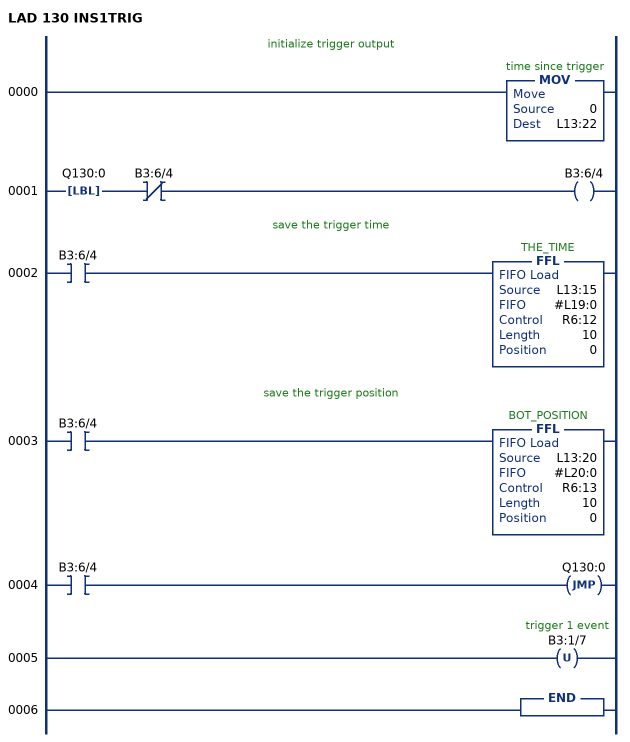
% Rung: 0 %
% initialize trigger output %
SOR MOV 0 L13:22 EOR
%   L13:22  "time since trigger" %
% Rung: 1 %
SOR LBL Q130:0 XIO B3:6/4 OTE B3:6/4 EOR
% Rung: 2 %
% save the trigger time %
SOR XIC B3:6/4 FFL L13:15 #L19:0 R6:12 10 0 EOR
%   L13:15  THE_TIME %
% Rung: 3 %
% save the trigger position %
SOR XIC B3:6/4 FFL L13:20 #L20:0 R6:13 10 0 EOR
%   L13:20  BOT_POSITION %
% Rung: 4 %
SOR XIC B3:6/4 JMP Q130:0 EOR
% Rung: 5 %
SOR OTU B3:1/7 EOR
%   B3:1/7  "trigger 1 event" %
% Rung: 6 %
SOR END EOR

LADDER 131 "XFER"
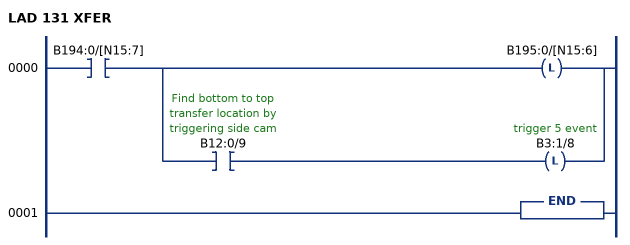
% Rung: 0 %
SOR XIC B194:0/[N15:7] BST OTL B195:0/[N15:6] NXB XIC B12:0/9 OTL B3:1/8 BND EOR
%   N15:7  XFER_OUT_LOC %
%   N15:6  XFER_IN_LOC %
%   B12:0/9  "Find bottom to top transfer location by triggering side cam" %
%   B3:1/8  "trigger 5 event" %
% Rung: 1 %
SOR END EOR

LADDER 140 "TOPOPTIC"
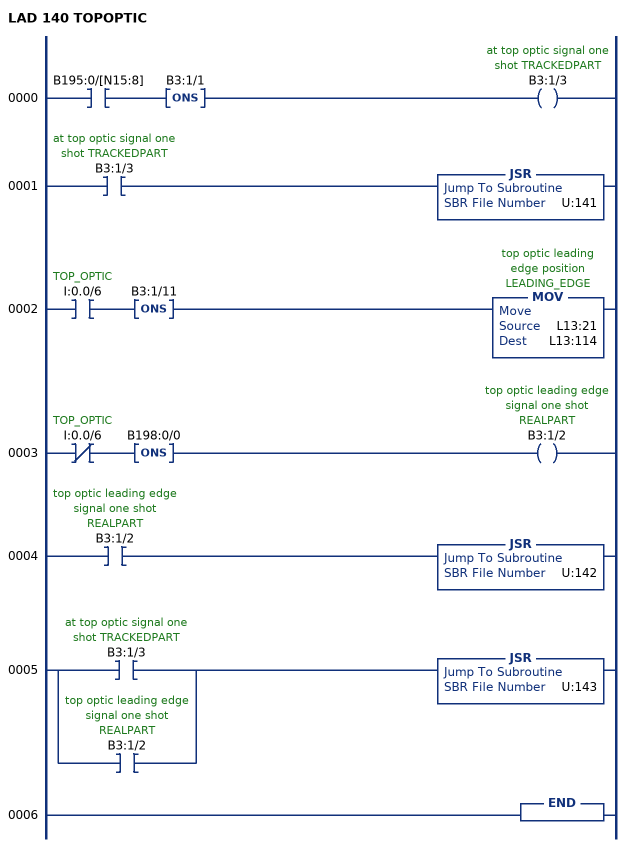
% Rung: 0 %
SOR XIC B195:0/[N15:8] ONS B3:1/1 OTE B3:1/3 EOR
%   N15:8  TOP_OPTIC_LOC %
%   B3:1/3  TRACKEDPART  "at top optic signal one shot" %
% Rung: 1 %
SOR XIC B3:1/3 JSR U:141 EOR
%   B3:1/3  TRACKEDPART  "at top optic signal one shot" %
% Rung: 2 %
SOR XIC I:0.0/6 ONS B3:1/11 MOV L13:21 L13:114 EOR
%   I:0.0/6  TOP_OPTIC %
%   L13:21  TOP_POSITION %
%   L13:114  LEADING_EDGE  "top optic leading edge position" %
% Rung: 3 %
SOR XIO I:0.0/6 ONS B198:0/0 OTE B3:1/2 EOR
%   I:0.0/6  TOP_OPTIC %
%   B3:1/2  REALPART  "top optic leading edge signal one shot" %
% Rung: 4 %
SOR XIC B3:1/2 JSR U:142 EOR
%   B3:1/2  REALPART  "top optic leading edge signal one shot" %
% Rung: 5 %
SOR BST XIC B3:1/3 NXB XIC B3:1/2 BND JSR U:143 EOR
%   B3:1/3  TRACKEDPART  "at top optic signal one shot" %
%   B3:1/2  REALPART  "top optic leading edge signal one shot" %
% Rung: 6 %
SOR END EOR

LADDER 141 "TOPOPVERT"
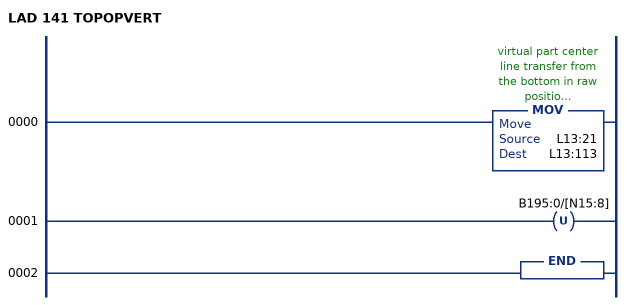
% Rung: 0 %
SOR MOV L13:21 L13:113 EOR
%   L13:21  TOP_POSITION %
%   L13:113  VERTUAL_PT_RAW_CL  "virtual part center line transfer from the bottom in raw position" %
% Rung: 1 %
SOR OTU B195:0/[N15:8] EOR
%   N15:8  TOP_OPTIC_LOC %
% Rung: 2 %
SOR END EOR

LADDER 142 "TOPOPREAL"
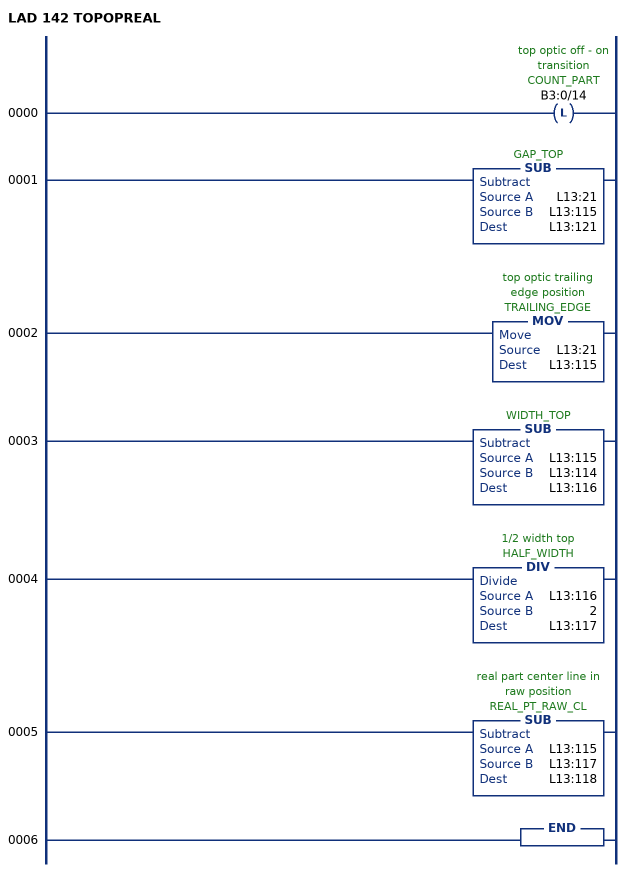
% Rung: 0 %
SOR OTL B3:0/14 EOR
%   B3:0/14  COUNT_PART  "top optic off - on transition" %
% Rung: 1 %
SOR SUB L13:21 L13:115 L13:121 EOR
%   L13:21  TOP_POSITION %
%   L13:115  TRAILING_EDGE  "top optic trailing edge position" %
%   L13:121  GAP_TOP %
% Rung: 2 %
SOR MOV L13:21 L13:115 EOR
%   L13:21  TOP_POSITION %
%   L13:115  TRAILING_EDGE  "top optic trailing edge position" %
% Rung: 3 %
SOR SUB L13:115 L13:114 L13:116 EOR
%   L13:115  TRAILING_EDGE  "top optic trailing edge position" %
%   L13:114  LEADING_EDGE  "top optic leading edge position" %
%   L13:116  WIDTH_TOP %
% Rung: 4 %
SOR DIV L13:116 2 L13:117 EOR
%   L13:116  WIDTH_TOP %
%   L13:117  HALF_WIDTH  "1/2 width top" %
% Rung: 5 %
SOR SUB L13:115 L13:117 L13:118 EOR
%   L13:115  TRAILING_EDGE  "top optic trailing edge position" %
%   L13:117  HALF_WIDTH  "1/2 width top" %
%   L13:118  REAL_PT_RAW_CL  "real part center line in raw position" %
% Rung: 6 %
SOR END EOR

LADDER 143 "TOPOPTEST"
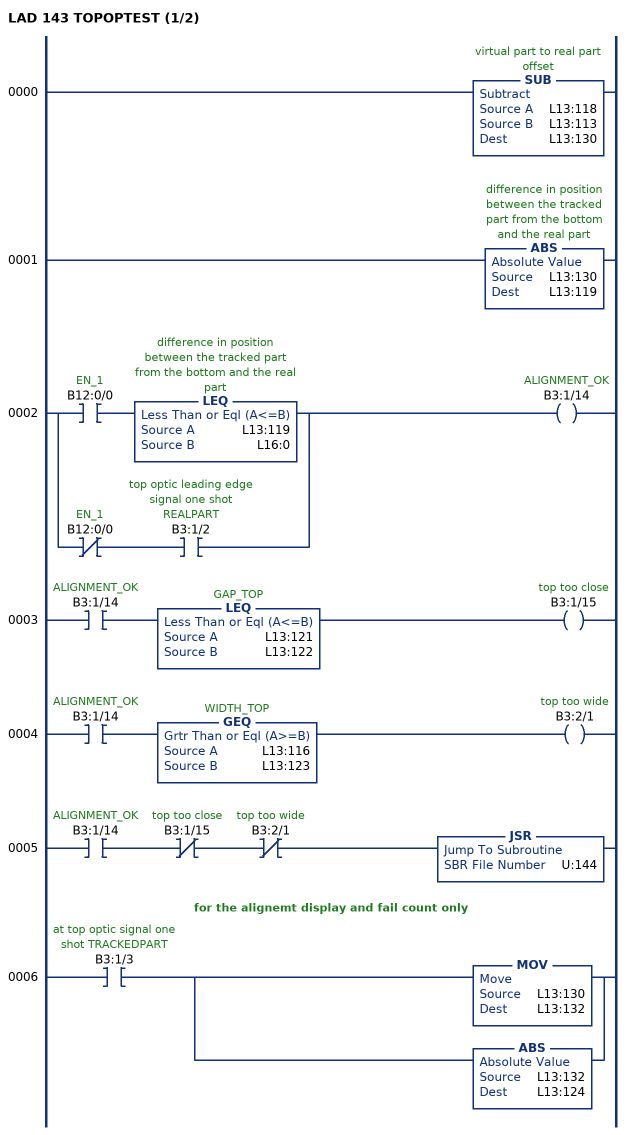
% Rung: 0 %
SOR SUB L13:118 L13:113 L13:130 EOR
%   L13:118  REAL_PT_RAW_CL  "real part center line in raw position" %
%   L13:113  VERTUAL_PT_RAW_CL  "virtual part center line transfer from the bottom in raw position" %
%   L13:130  "virtual part to real part offset" %
% Rung: 1 %
SOR ABS L13:130 L13:119 EOR
%   L13:130  "virtual part to real part offset" %
%   L13:119  "difference in position between the tracked part from the bottom and the real part" %
% Rung: 2 %
SOR BST XIC B12:0/0 LEQ L13:119 L16:0 NXB XIO B12:0/0 XIC B3:1/2 BND OTE B3:1/14 EOR
%   B12:0/0  EN_1 %
%   L13:119  "difference in position between the tracked part from the bottom and the real part" %
%   L16:0  MAX_OFFSET %
%   B3:1/2  REALPART  "top optic leading edge signal one shot" %
%   B3:1/14  ALIGNMENT_OK %
% Rung: 3 %
SOR XIC B3:1/14 LEQ L13:121 L13:122 OTE B3:1/15 EOR
%   B3:1/14  ALIGNMENT_OK %
%   L13:121  GAP_TOP %
%   L13:122  MIN_GAP_TOP %
%   B3:1/15  "top too close" %
% Rung: 4 %
SOR XIC B3:1/14 GEQ L13:116 L13:123 OTE B3:2/1 EOR
%   B3:1/14  ALIGNMENT_OK %
%   L13:116  WIDTH_TOP %
%   L13:123  MAX_WIDTH_TOP %
%   B3:2/1  "top too wide" %
% Rung: 5 %
SOR XIC B3:1/14 XIO B3:1/15 XIO B3:2/1 JSR U:144 EOR
%   B3:1/14  ALIGNMENT_OK %
%   B3:1/15  "top too close" %
%   B3:2/1  "top too wide" %
% Rung: 6 %
% TITLE: for the alignemt display and fail count only %
SOR XIC B3:1/3 BST MOV L13:130 L13:132 NXB ABS L13:132 L13:124 BND EOR
%   B3:1/3  TRACKEDPART  "at top optic signal one shot" %
%   L13:130  "virtual part to real part offset" %

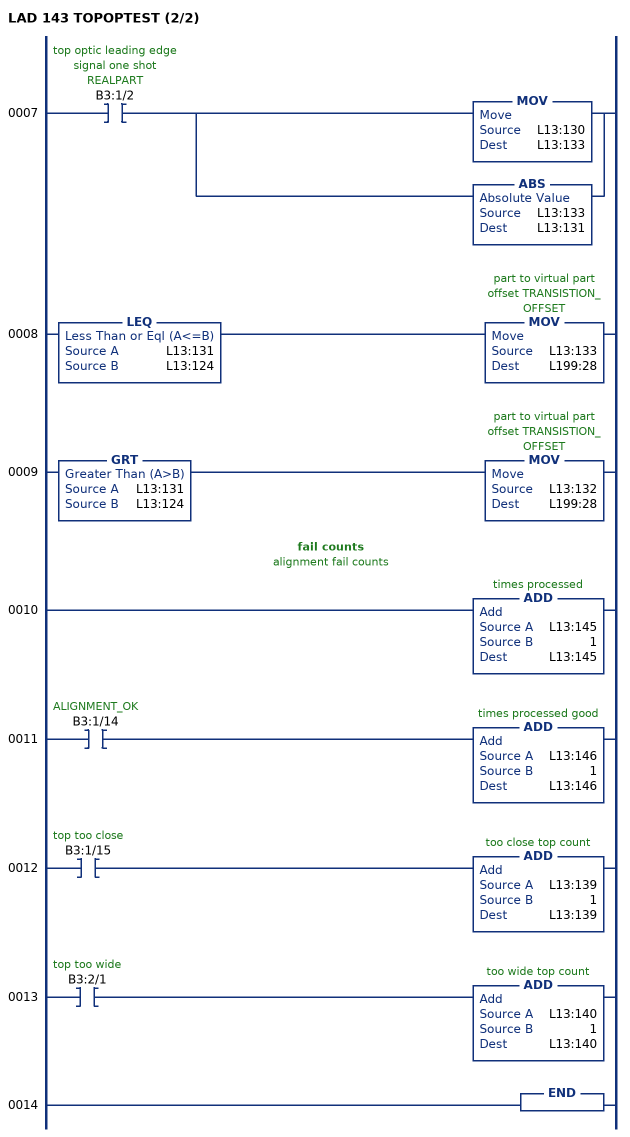
% Rung: 7 %
SOR XIC B3:1/2 BST MOV L13:130 L13:133 NXB ABS L13:133 L13:131 BND EOR
%   B3:1/2  REALPART  "top optic leading edge signal one shot" %
%   L13:130  "virtual part to real part offset" %
% Rung: 8 %
SOR LEQ L13:131 L13:124 MOV L13:133 L199:28 EOR
%   L199:28  TRANSISTION_OFFSET  "part to virtual part offset" %
% Rung: 9 %
SOR GRT L13:131 L13:124 MOV L13:132 L199:28 EOR
%   L199:28  TRANSISTION_OFFSET  "part to virtual part offset" %
% Rung: 10 %
% TITLE: fail counts %
% alignment fail counts %
SOR ADD L13:145 1 L13:145 EOR
%   L13:145  "times processed" %
% Rung: 11 %
SOR XIC B3:1/14 ADD L13:146 1 L13:146 EOR
%   B3:1/14  ALIGNMENT_OK %
%   L13:146  "times processed good" %
% Rung: 12 %
SOR XIC B3:1/15 ADD L13:139 1 L13:139 EOR
%   B3:1/15  "top too close" %
%   L13:139  "too close top count" %
% Rung: 13 %
SOR XIC B3:2/1 ADD L13:140 1 L13:140 EOR
%   B3:2/1  "top too wide" %
%   L13:140  "too wide top count" %
% Rung: 14 %
SOR END EOR

LADDER 144 "TOPOPOKAY"
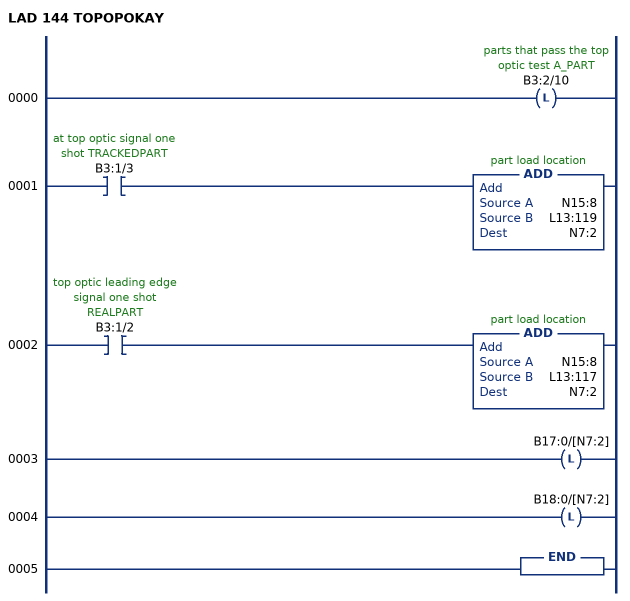
% Rung: 0 %
SOR OTL B3:2/10 EOR
%   B3:2/10  A_PART  "parts that pass the top optic test" %
% Rung: 1 %
SOR XIC B3:1/3 ADD N15:8 L13:119 N7:2 EOR
%   B3:1/3  TRACKEDPART  "at top optic signal one shot" %
%   N15:8  TOP_OPTIC_LOC %
%   L13:119  "difference in position between the tracked part from the bottom and the real part" %
%   N7:2  "part load location" %
% Rung: 2 %
SOR XIC B3:1/2 ADD N15:8 L13:117 N7:2 EOR
%   B3:1/2  REALPART  "top optic leading edge signal one shot" %
%   N15:8  TOP_OPTIC_LOC %
%   L13:117  HALF_WIDTH  "1/2 width top" %
%   N7:2  "part load location" %
% Rung: 3 %
SOR OTL B17:0/[N7:2] EOR
%   N7:2  "part load location" %
% Rung: 4 %
SOR OTL B18:0/[N7:2] EOR
%   N7:2  "part load location" %
% Rung: 5 %
SOR END EOR

LADDER 149 "INS5RESULT"
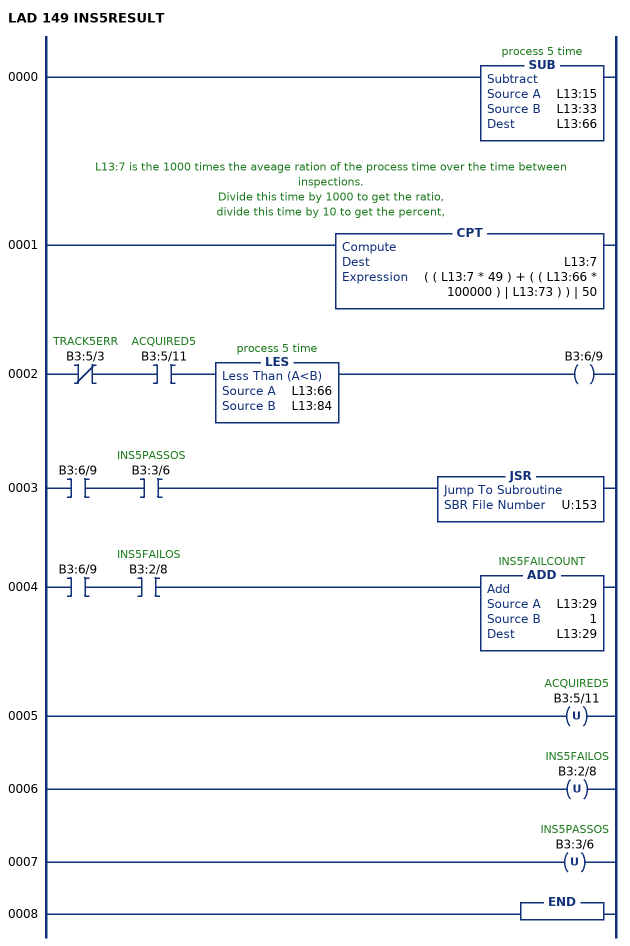
% Rung: 0 %
SOR SUB L13:15 L13:33 L13:66 EOR
%   L13:15  THE_TIME %
%   L13:33  TIMEOFACQ5  "the time of the last acquire" %
%   L13:66  "process 5 time" %
% Rung: 1 %
% L13:7 is the 1000 times the aveage ration of the process time over the time between inspections.
% Divide this time by 1000 to get the ratio,
% divide this time by 10 to get the percent, %
SOR CPT L13:7 " ( ( L13:7 * 49 ) + ( ( L13:66 * 100000 ) | L13:73 ) ) | 50 " EOR
%   L13:66  "process 5 time" %
%   L13:73  TBI %
% Rung: 2 %
SOR XIO B3:5/3 XIC B3:5/11 LES L13:66 L13:84 OTE B3:6/9 EOR
%   B3:5/3  TRACK5ERR %
%   B3:5/11  ACQUIRED5 %
%   L13:66  "process 5 time" %
% Rung: 3 %
SOR XIC B3:6/9 XIC B3:3/6 JSR U:153 EOR
%   B3:3/6  INS5PASSOS %
% Rung: 4 %
SOR XIC B3:6/9 XIC B3:2/8 ADD L13:29 1 L13:29 EOR
%   B3:2/8  INS5FAILOS %
%   L13:29  INS5FAILCOUNT %
% Rung: 5 %
SOR OTU B3:5/11 EOR
%   B3:5/11  ACQUIRED5 %
% Rung: 6 %
SOR OTU B3:2/8 EOR
%   B3:2/8  INS5FAILOS %
% Rung: 7 %
SOR OTU B3:3/6 EOR
%   B3:3/6  INS5PASSOS %
% Rung: 8 %
SOR END EOR

LADDER 150 "FIXERR5"
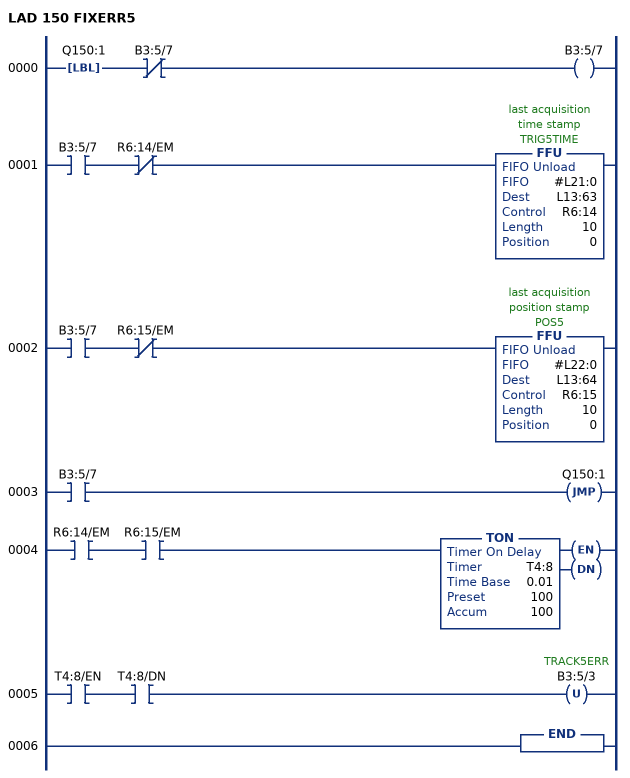
% Rung: 0 %
SOR LBL Q150:1 XIO B3:5/7 OTE B3:5/7 EOR
% Rung: 1 %
SOR XIC B3:5/7 XIO R6:14/EM FFU #L21:0 L13:63 R6:14 10 0 EOR
%   L13:63  TRIG5TIME  "last acquisition time stamp" %
% Rung: 2 %
SOR XIC B3:5/7 XIO R6:15/EM FFU #L22:0 L13:64 R6:15 10 0 EOR
%   L13:64  POS5  "last acquisition position stamp" %
% Rung: 3 %
SOR XIC B3:5/7 JMP Q150:1 EOR
% Rung: 4 %
SOR XIC R6:14/EM XIC R6:15/EM TON T4:8 0.01 100 100 EOR
% Rung: 5 %
SOR XIC T4:8/EN XIC T4:8/DN OTU B3:5/3 EOR
%   B3:5/3  TRACK5ERR %
% Rung: 6 %
SOR END EOR

LADDER 152 "INS5"
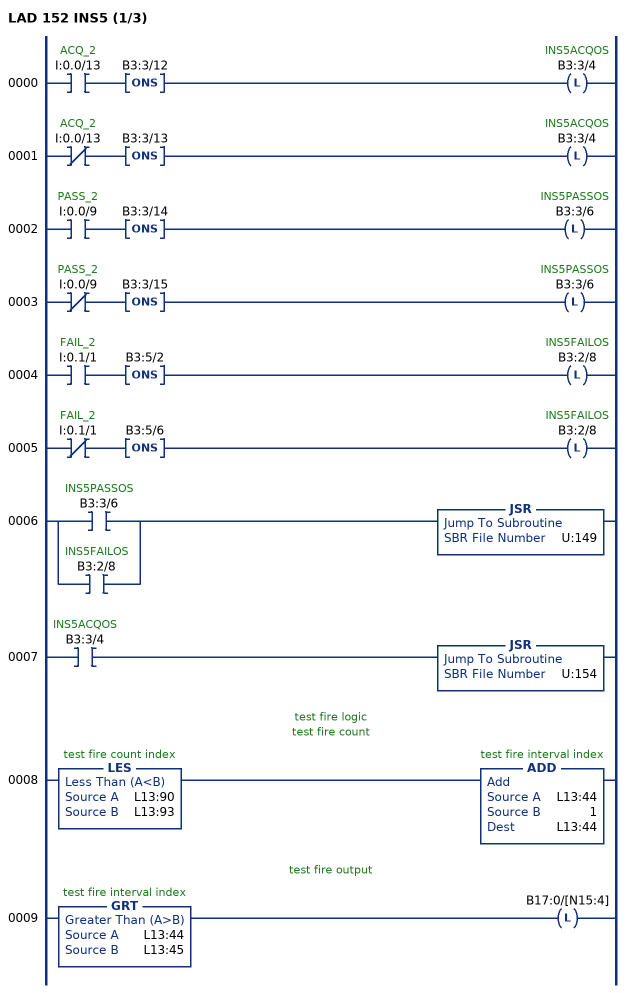
% Rung: 0 %
SOR XIC I:0.0/13 ONS B3:3/12 OTL B3:3/4 EOR
%   I:0.0/13  ACQ_2 %
%   B3:3/4  INS5ACQOS %
% Rung: 1 %
SOR XIO I:0.0/13 ONS B3:3/13 OTL B3:3/4 EOR
%   I:0.0/13  ACQ_2 %
%   B3:3/4  INS5ACQOS %
% Rung: 2 %
SOR XIC I:0.0/9 ONS B3:3/14 OTL B3:3/6 EOR
%   I:0.0/9  PASS_2 %
%   B3:3/6  INS5PASSOS %
% Rung: 3 %
SOR XIO I:0.0/9 ONS B3:3/15 OTL B3:3/6 EOR
%   I:0.0/9  PASS_2 %
%   B3:3/6  INS5PASSOS %
% Rung: 4 %
SOR XIC I:0.1/1 ONS B3:5/2 OTL B3:2/8 EOR
%   I:0.1/1  FAIL_2 %
%   B3:2/8  INS5FAILOS %
% Rung: 5 %
SOR XIO I:0.1/1 ONS B3:5/6 OTL B3:2/8 EOR
%   I:0.1/1  FAIL_2 %
%   B3:2/8  INS5FAILOS %
% Rung: 6 %
SOR BST XIC B3:3/6 NXB XIC B3:2/8 BND JSR U:149 EOR
%   B3:3/6  INS5PASSOS %
%   B3:2/8  INS5FAILOS %
% Rung: 7 %
SOR XIC B3:3/4 JSR U:154 EOR
%   B3:3/4  INS5ACQOS %
% Rung: 8 %
% test fire logic
% 
% test fire count %
SOR LES L13:90 L13:93 ADD L13:44 1 L13:44 EOR
%   L13:90  "test fire count index" %
%   L13:93  "test fire count" %
%   L13:44  "test fire interval index" %
% Rung: 9 %
% test fire output %
SOR GRT L13:44 L13:45 OTL B17:0/[N15:4] EOR
%   L13:44  "test fire interval index" %
%   L13:45  "test fire interval" %
%   N15:4  INS_5_TRIG_LOC %

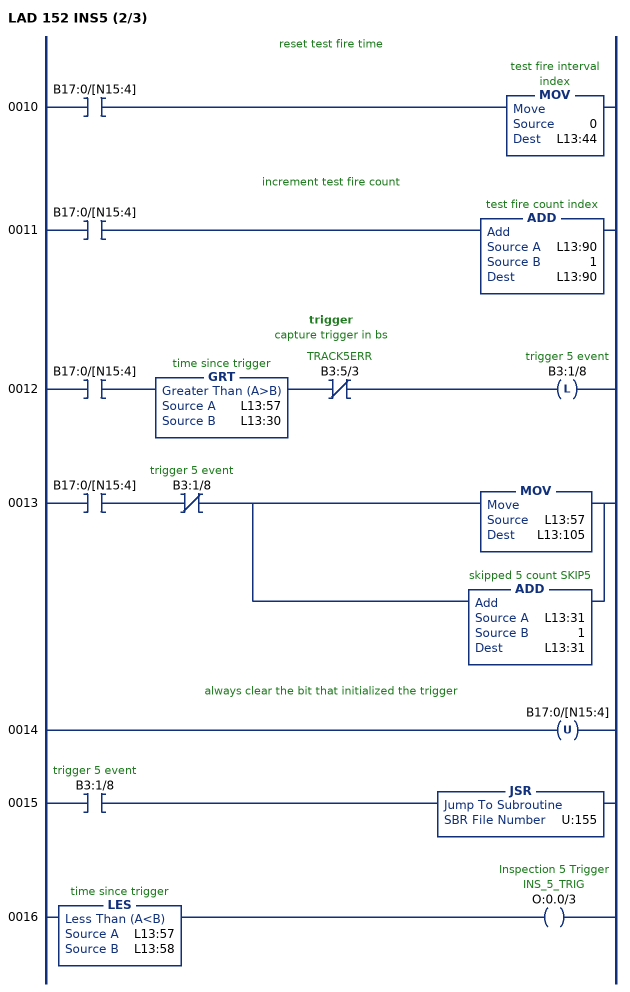
% Rung: 10 %
% reset test fire time %
SOR XIC B17:0/[N15:4] MOV 0 L13:44 EOR
%   N15:4  INS_5_TRIG_LOC %
%   L13:44  "test fire interval index" %
% Rung: 11 %
% increment test fire count %
SOR XIC B17:0/[N15:4] ADD L13:90 1 L13:90 EOR
%   N15:4  INS_5_TRIG_LOC %
%   L13:90  "test fire count index" %
% Rung: 12 %
% TITLE: trigger %
% capture trigger in bs %
SOR XIC B17:0/[N15:4] GRT L13:57 L13:30 XIO B3:5/3 OTL B3:1/8 EOR
%   N15:4  INS_5_TRIG_LOC %
%   L13:57  "time since trigger" %
%   B3:5/3  TRACK5ERR %
%   B3:1/8  "trigger 5 event" %
% Rung: 13 %
SOR XIC B17:0/[N15:4] XIO B3:1/8 BST MOV L13:57 L13:105 NXB ADD L13:31 1 L13:31 BND EOR
%   N15:4  INS_5_TRIG_LOC %
%   B3:1/8  "trigger 5 event" %
%   L13:57  "time since trigger" %
%   L13:31  SKIP5  "skipped 5 count" %
% Rung: 14 %
% always clear the bit that initialized the trigger %
SOR OTU B17:0/[N15:4] EOR
%   N15:4  INS_5_TRIG_LOC %
% Rung: 15 %
SOR XIC B3:1/8 JSR U:155 EOR
%   B3:1/8  "trigger 5 event" %
% Rung: 16 %
SOR LES L13:57 L13:58 OTE O:0.0/3 EOR
%   L13:57  "time since trigger" %
%   O:0.0/3  INS_5_TRIG  "Inspection 5 Trigger" %

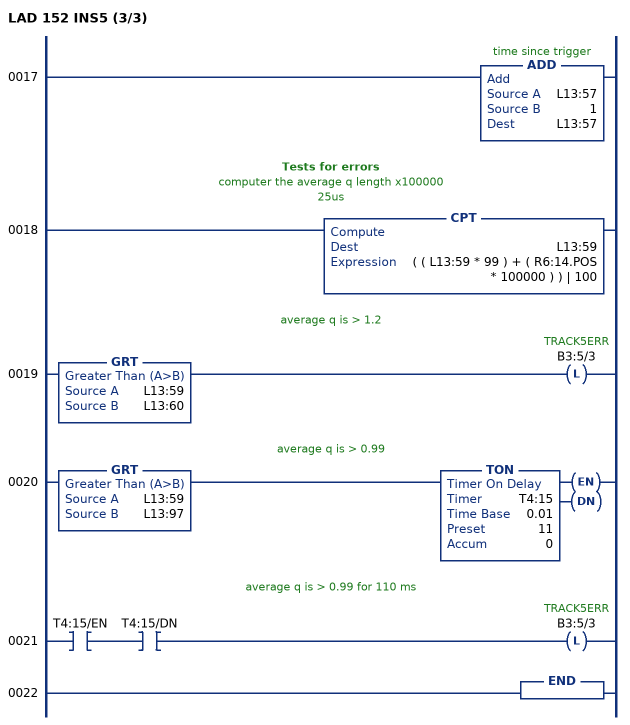
% Rung: 17 %
SOR ADD L13:57 1 L13:57 EOR
%   L13:57  "time since trigger" %
% Rung: 18 %
% TITLE: Tests for errors %
% computer the average q length x100000
% 25us %
SOR CPT L13:59 " ( ( L13:59 * 99 ) + ( R6:14.POS * 100000 ) ) | 100 " EOR
% Rung: 19 %
% average q is > 1.2 %
SOR GRT L13:59 L13:60 OTL B3:5/3 EOR
%   B3:5/3  TRACK5ERR %
% Rung: 20 %
% average q is > 0.99 %
SOR GRT L13:59 L13:97 TON T4:15 0.01 11 0 EOR
% Rung: 21 %
% average q is > 0.99 for 110 ms %
SOR XIC T4:15/EN XIC T4:15/DN OTL B3:5/3 EOR
%   B3:5/3  TRACK5ERR %
% Rung: 22 %
SOR END EOR

LADDER 153 "INS5PASS"
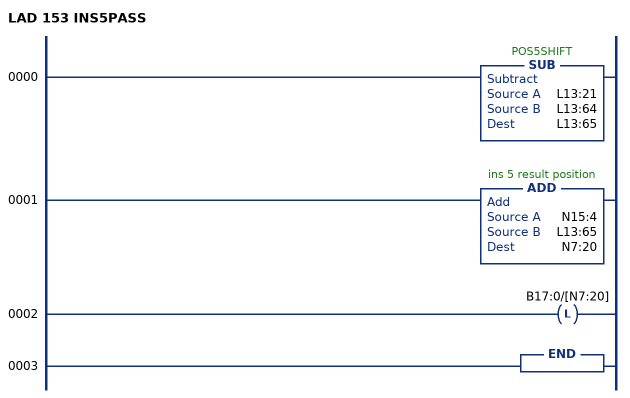
% Rung: 0 %
SOR SUB L13:21 L13:64 L13:65 EOR
%   L13:21  TOP_POSITION %
%   L13:64  POS5  "last acquisition position stamp" %
%   L13:65  POS5SHIFT %
% Rung: 1 %
SOR ADD N15:4 L13:65 N7:20 EOR
%   N15:4  INS_5_TRIG_LOC %
%   L13:65  POS5SHIFT %
%   N7:20  "ins 5 result position" %
% Rung: 2 %
SOR OTL B17:0/[N7:20] EOR
%   N7:20  "ins 5 result position" %
% Rung: 3 %
SOR END EOR

LADDER 154 "INS5ACQ"
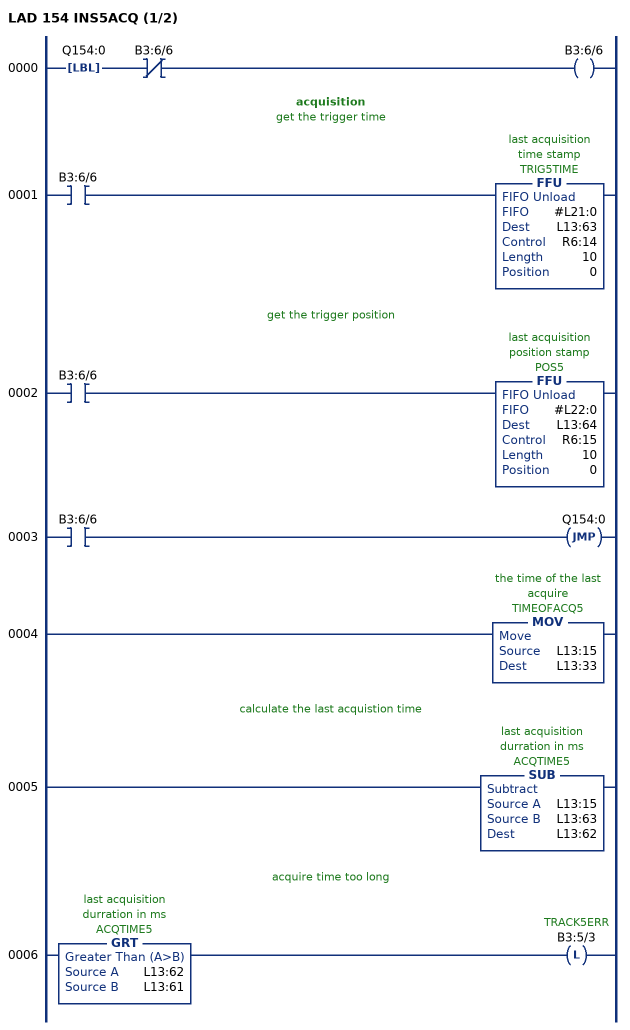
% Rung: 0 %
SOR LBL Q154:0 XIO B3:6/6 OTE B3:6/6 EOR
% Rung: 1 %
% TITLE: acquisition %
% get the trigger time %
SOR XIC B3:6/6 FFU #L21:0 L13:63 R6:14 10 0 EOR
%   L13:63  TRIG5TIME  "last acquisition time stamp" %
% Rung: 2 %
% get the trigger position %
SOR XIC B3:6/6 FFU #L22:0 L13:64 R6:15 10 0 EOR
%   L13:64  POS5  "last acquisition position stamp" %
% Rung: 3 %
SOR XIC B3:6/6 JMP Q154:0 EOR
% Rung: 4 %
SOR MOV L13:15 L13:33 EOR
%   L13:15  THE_TIME %
%   L13:33  TIMEOFACQ5  "the time of the last acquire" %
% Rung: 5 %
% calculate the last acquistion time %
SOR SUB L13:15 L13:63 L13:62 EOR
%   L13:15  THE_TIME %
%   L13:63  TRIG5TIME  "last acquisition time stamp" %
%   L13:62  ACQTIME5  "last acquisition durration in ms" %
% Rung: 6 %
% acquire time too long %
SOR GRT L13:62 L13:61 OTL B3:5/3 EOR
%   L13:62  ACQTIME5  "last acquisition durration in ms" %
%   L13:61  "max acquisition time in ms" %
%   B3:5/3  TRACK5ERR %

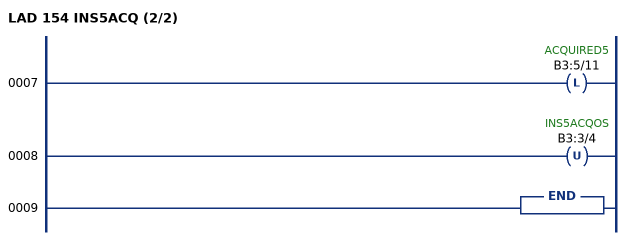
% Rung: 7 %
SOR OTL B3:5/11 EOR
%   B3:5/11  ACQUIRED5 %
% Rung: 8 %
SOR OTU B3:3/4 EOR
%   B3:3/4  INS5ACQOS %
% Rung: 9 %
SOR END EOR

LADDER 155 "INS5TRIG"
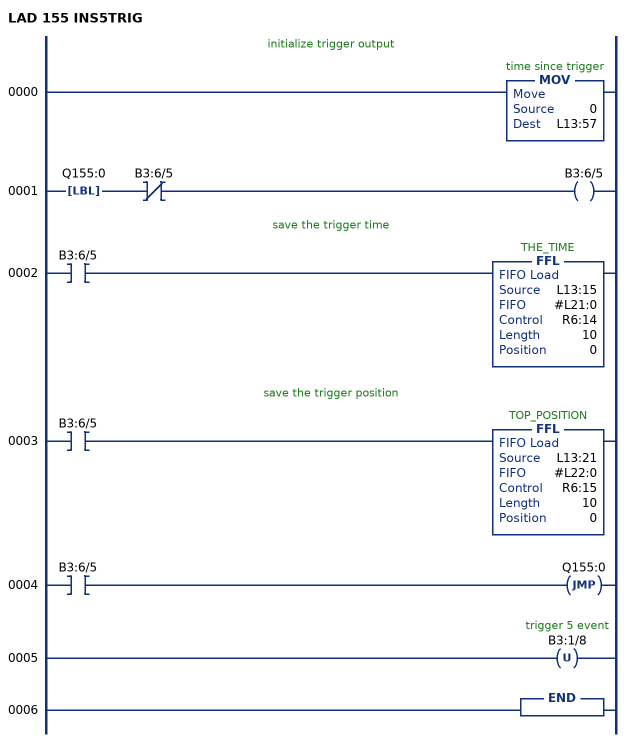
% Rung: 0 %
% initialize trigger output %
SOR MOV 0 L13:57 EOR
%   L13:57  "time since trigger" %
% Rung: 1 %
SOR LBL Q155:0 XIO B3:6/5 OTE B3:6/5 EOR
% Rung: 2 %
% save the trigger time %
SOR XIC B3:6/5 FFL L13:15 #L21:0 R6:14 10 0 EOR
%   L13:15  THE_TIME %
% Rung: 3 %
% save the trigger position %
SOR XIC B3:6/5 FFL L13:21 #L22:0 R6:15 10 0 EOR
%   L13:21  TOP_POSITION %
% Rung: 4 %
SOR XIC B3:6/5 JMP Q155:0 EOR
% Rung: 5 %
SOR OTU B3:1/8 EOR
%   B3:1/8  "trigger 5 event" %
% Rung: 6 %
SOR END EOR

LADDER 159 "INS6RESULT"
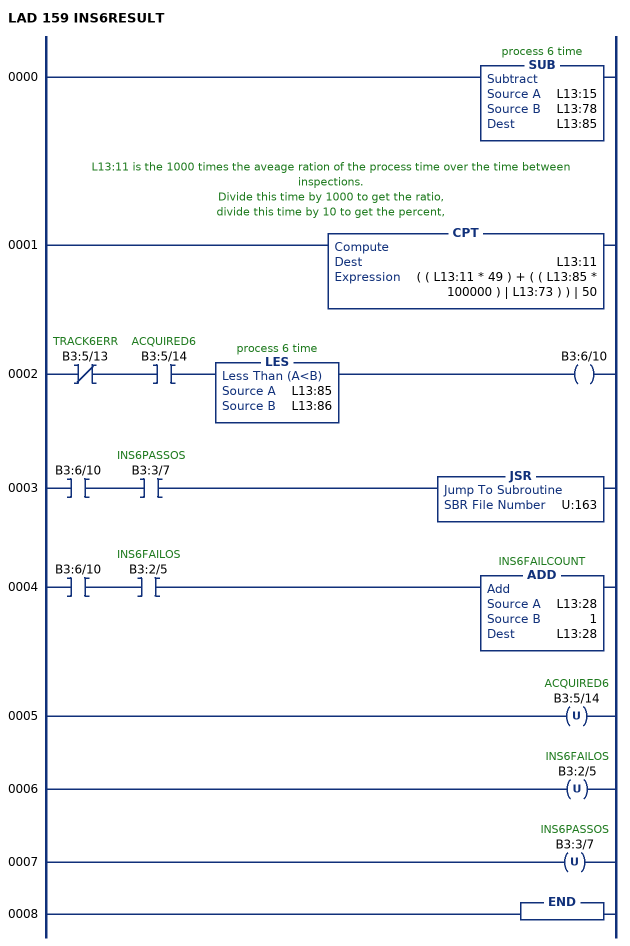
% Rung: 0 %
SOR SUB L13:15 L13:78 L13:85 EOR
%   L13:15  THE_TIME %
%   L13:78  TIMEOFACQ6  "the time of the last acquire" %
%   L13:85  "process 6 time" %
% Rung: 1 %
% L13:11 is the 1000 times the aveage ration of the process time over the time between inspections.
% Divide this time by 1000 to get the ratio,
% divide this time by 10 to get the percent, %
SOR CPT L13:11 " ( ( L13:11 * 49 ) + ( ( L13:85 * 100000 ) | L13:73 ) ) | 50 " EOR
%   L13:85  "process 6 time" %
%   L13:73  TBI %
% Rung: 2 %
SOR XIO B3:5/13 XIC B3:5/14 LES L13:85 L13:86 OTE B3:6/10 EOR
%   B3:5/13  TRACK6ERR %
%   B3:5/14  ACQUIRED6 %
%   L13:85  "process 6 time" %
% Rung: 3 %
SOR XIC B3:6/10 XIC B3:3/7 JSR U:163 EOR
%   B3:3/7  INS6PASSOS %
% Rung: 4 %
SOR XIC B3:6/10 XIC B3:2/5 ADD L13:28 1 L13:28 EOR
%   B3:2/5  INS6FAILOS %
%   L13:28  INS6FAILCOUNT %
% Rung: 5 %
SOR OTU B3:5/14 EOR
%   B3:5/14  ACQUIRED6 %
% Rung: 6 %
SOR OTU B3:2/5 EOR
%   B3:2/5  INS6FAILOS %
% Rung: 7 %
SOR OTU B3:3/7 EOR
%   B3:3/7  INS6PASSOS %
% Rung: 8 %
SOR END EOR

LADDER 160 "FIXERR6"
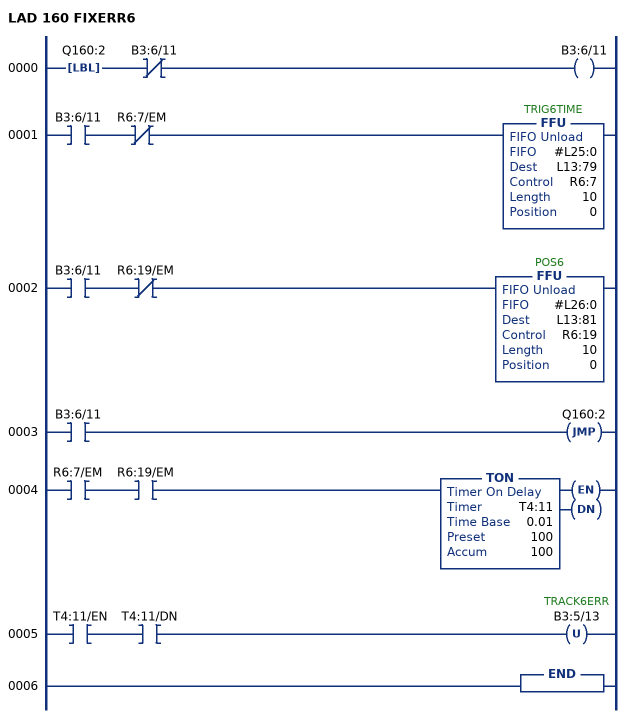
% Rung: 0 %
SOR LBL Q160:2 XIO B3:6/11 OTE B3:6/11 EOR
% Rung: 1 %
SOR XIC B3:6/11 XIO R6:7/EM FFU #L25:0 L13:79 R6:7 10 0 EOR
%   L13:79  TRIG6TIME %
% Rung: 2 %
SOR XIC B3:6/11 XIO R6:19/EM FFU #L26:0 L13:81 R6:19 10 0 EOR
%   L13:81  POS6 %
% Rung: 3 %
SOR XIC B3:6/11 JMP Q160:2 EOR
% Rung: 4 %
SOR XIC R6:7/EM XIC R6:19/EM TON T4:11 0.01 100 100 EOR
% Rung: 5 %
SOR XIC T4:11/EN XIC T4:11/DN OTU B3:5/13 EOR
%   B3:5/13  TRACK6ERR %
% Rung: 6 %
SOR END EOR

LADDER 162 "INS6"
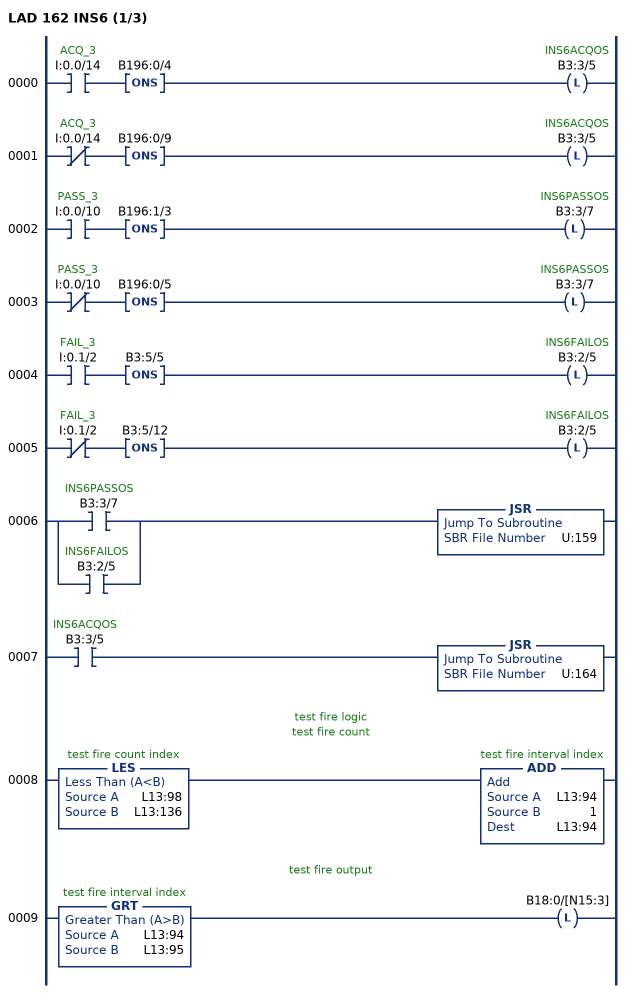
% Rung: 0 %
SOR XIC I:0.0/14 ONS B196:0/4 OTL B3:3/5 EOR
%   I:0.0/14  ACQ_3 %
%   B3:3/5  INS6ACQOS %
% Rung: 1 %
SOR XIO I:0.0/14 ONS B196:0/9 OTL B3:3/5 EOR
%   I:0.0/14  ACQ_3 %
%   B3:3/5  INS6ACQOS %
% Rung: 2 %
SOR XIC I:0.0/10 ONS B196:1/3 OTL B3:3/7 EOR
%   I:0.0/10  PASS_3 %
%   B3:3/7  INS6PASSOS %
% Rung: 3 %
SOR XIO I:0.0/10 ONS B196:0/5 OTL B3:3/7 EOR
%   I:0.0/10  PASS_3 %
%   B3:3/7  INS6PASSOS %
% Rung: 4 %
SOR XIC I:0.1/2 ONS B3:5/5 OTL B3:2/5 EOR
%   I:0.1/2  FAIL_3 %
%   B3:2/5  INS6FAILOS %
% Rung: 5 %
SOR XIO I:0.1/2 ONS B3:5/12 OTL B3:2/5 EOR
%   I:0.1/2  FAIL_3 %
%   B3:2/5  INS6FAILOS %
% Rung: 6 %
SOR BST XIC B3:3/7 NXB XIC B3:2/5 BND JSR U:159 EOR
%   B3:3/7  INS6PASSOS %
%   B3:2/5  INS6FAILOS %
% Rung: 7 %
SOR XIC B3:3/5 JSR U:164 EOR
%   B3:3/5  INS6ACQOS %
% Rung: 8 %
% test fire logic
% 
% test fire count %
SOR LES L13:98 L13:136 ADD L13:94 1 L13:94 EOR
%   L13:98  "test fire count index" %
%   L13:136  "test fire count" %
%   L13:94  "test fire interval index" %
% Rung: 9 %
% test fire output %
SOR GRT L13:94 L13:95 OTL B18:0/[N15:3] EOR
%   L13:94  "test fire interval index" %
%   L13:95  "test fire interval" %
%   N15:3  INS_6_TRIG_LOC %

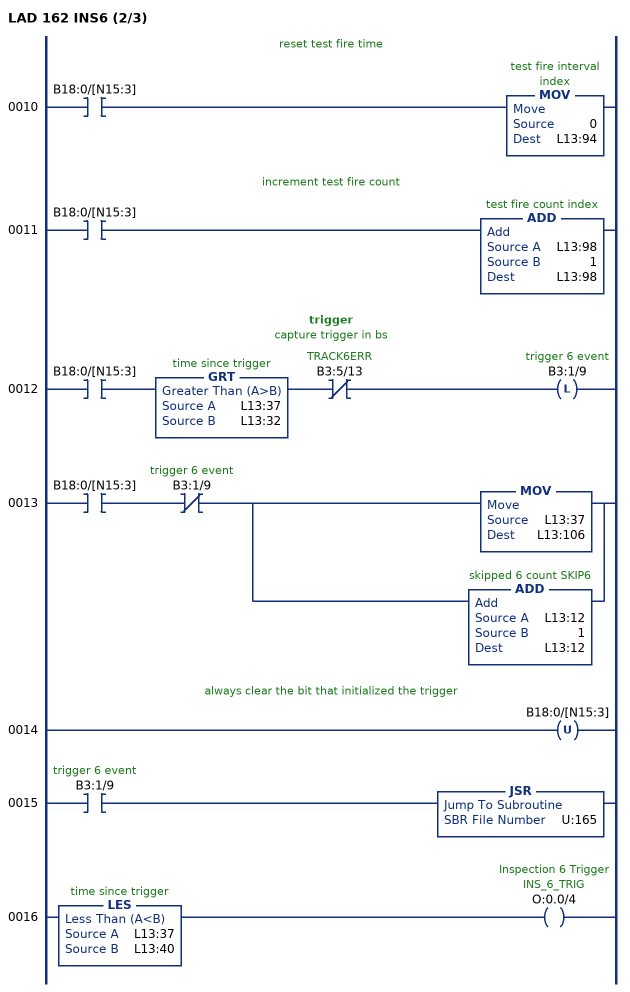
% Rung: 10 %
% reset test fire time %
SOR XIC B18:0/[N15:3] MOV 0 L13:94 EOR
%   N15:3  INS_6_TRIG_LOC %
%   L13:94  "test fire interval index" %
% Rung: 11 %
% increment test fire count %
SOR XIC B18:0/[N15:3] ADD L13:98 1 L13:98 EOR
%   N15:3  INS_6_TRIG_LOC %
%   L13:98  "test fire count index" %
% Rung: 12 %
% TITLE: trigger %
% capture trigger in bs %
SOR XIC B18:0/[N15:3] GRT L13:37 L13:32 XIO B3:5/13 OTL B3:1/9 EOR
%   N15:3  INS_6_TRIG_LOC %
%   L13:37  "time since trigger" %
%   B3:5/13  TRACK6ERR %
%   B3:1/9  "trigger 6 event" %
% Rung: 13 %
SOR XIC B18:0/[N15:3] XIO B3:1/9 BST MOV L13:37 L13:106 NXB ADD L13:12 1 L13:12 BND EOR
%   N15:3  INS_6_TRIG_LOC %
%   B3:1/9  "trigger 6 event" %
%   L13:37  "time since trigger" %
%   L13:12  SKIP6  "skipped 6 count" %
% Rung: 14 %
% always clear the bit that initialized the trigger %
SOR OTU B18:0/[N15:3] EOR
%   N15:3  INS_6_TRIG_LOC %
% Rung: 15 %
SOR XIC B3:1/9 JSR U:165 EOR
%   B3:1/9  "trigger 6 event" %
% Rung: 16 %
SOR LES L13:37 L13:40 OTE O:0.0/4 EOR
%   L13:37  "time since trigger" %
%   L13:40  "last part time" %
%   O:0.0/4  INS_6_TRIG  "Inspection 6 Trigger" %

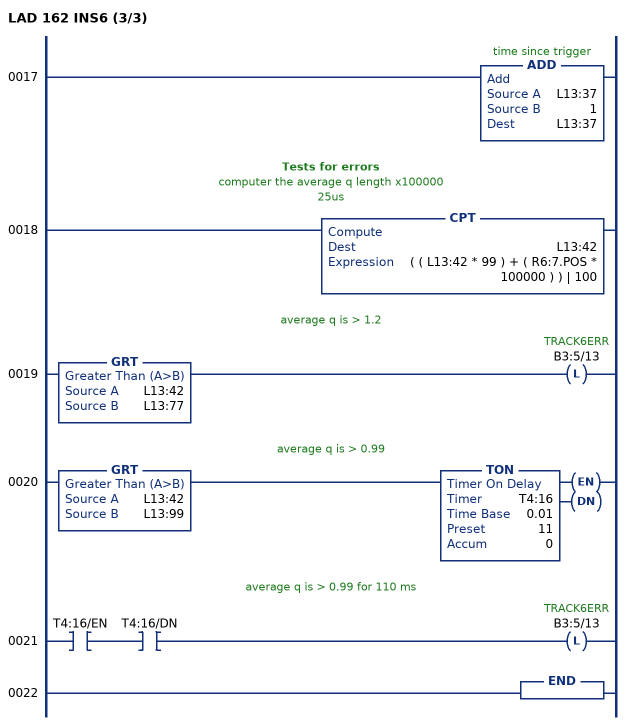
% Rung: 17 %
SOR ADD L13:37 1 L13:37 EOR
%   L13:37  "time since trigger" %
% Rung: 18 %
% TITLE: Tests for errors %
% computer the average q length x100000
% 25us %
SOR CPT L13:42 " ( ( L13:42 * 99 ) + ( R6:7.POS * 100000 ) ) | 100 " EOR
% Rung: 19 %
% average q is > 1.2 %
SOR GRT L13:42 L13:77 OTL B3:5/13 EOR
%   B3:5/13  TRACK6ERR %
% Rung: 20 %
% average q is > 0.99 %
SOR GRT L13:42 L13:99 TON T4:16 0.01 11 0 EOR
% Rung: 21 %
% average q is > 0.99 for 110 ms %
SOR XIC T4:16/EN XIC T4:16/DN OTL B3:5/13 EOR
%   B3:5/13  TRACK6ERR %
% Rung: 22 %
SOR END EOR

LADDER 163 "INS6PASS"
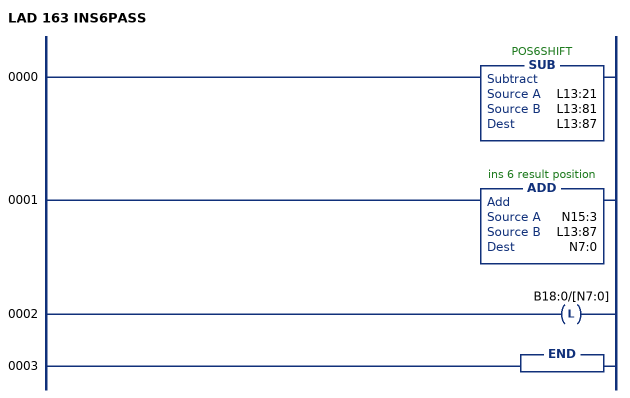
% Rung: 0 %
SOR SUB L13:21 L13:81 L13:87 EOR
%   L13:21  TOP_POSITION %
%   L13:81  POS6 %
%   L13:87  POS6SHIFT %
% Rung: 1 %
SOR ADD N15:3 L13:87 N7:0 EOR
%   N15:3  INS_6_TRIG_LOC %
%   L13:87  POS6SHIFT %
%   N7:0  "ins 6 result position" %
% Rung: 2 %
SOR OTL B18:0/[N7:0] EOR
%   N7:0  "ins 6 result position" %
% Rung: 3 %
SOR END EOR

LADDER 164 "INS6ACQ"
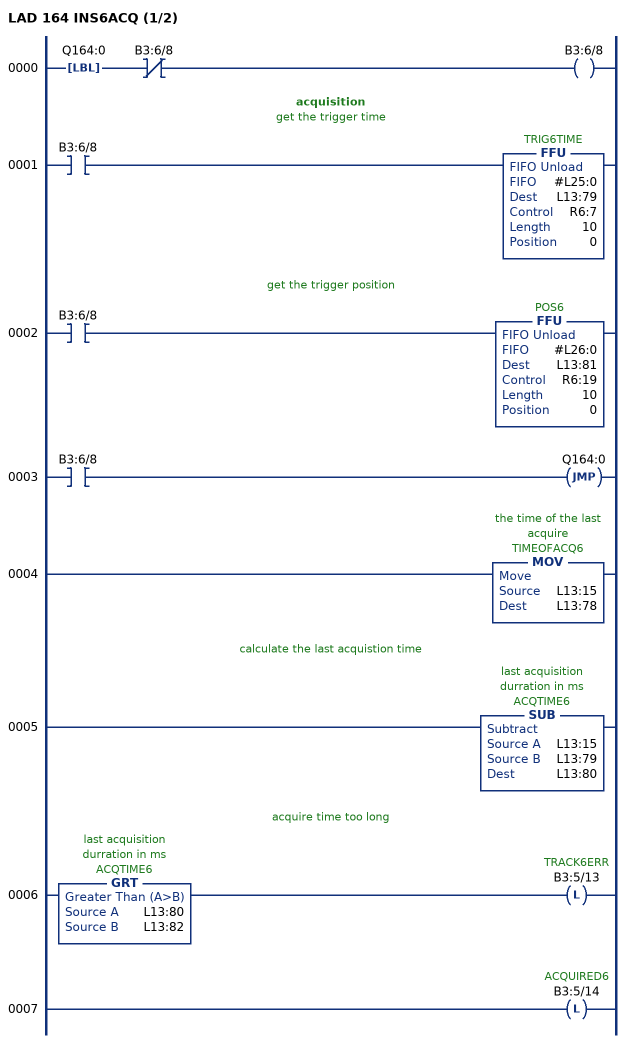
% Rung: 0 %
SOR LBL Q164:0 XIO B3:6/8 OTE B3:6/8 EOR
% Rung: 1 %
% TITLE: acquisition %
% get the trigger time %
SOR XIC B3:6/8 FFU #L25:0 L13:79 R6:7 10 0 EOR
%   L13:79  TRIG6TIME %
% Rung: 2 %
% get the trigger position %
SOR XIC B3:6/8 FFU #L26:0 L13:81 R6:19 10 0 EOR
%   L13:81  POS6 %
% Rung: 3 %
SOR XIC B3:6/8 JMP Q164:0 EOR
% Rung: 4 %
SOR MOV L13:15 L13:78 EOR
%   L13:15  THE_TIME %
%   L13:78  TIMEOFACQ6  "the time of the last acquire" %
% Rung: 5 %
% calculate the last acquistion time %
SOR SUB L13:15 L13:79 L13:80 EOR
%   L13:15  THE_TIME %
%   L13:79  TRIG6TIME %
%   L13:80  ACQTIME6  "last acquisition durration in ms" %
% Rung: 6 %
% acquire time too long %
SOR GRT L13:80 L13:82 OTL B3:5/13 EOR
%   L13:80  ACQTIME6  "last acquisition durration in ms" %
%   B3:5/13  TRACK6ERR %
% Rung: 7 %
SOR OTL B3:5/14 EOR
%   B3:5/14  ACQUIRED6 %

